TYPE EL3002_DEV_STATUS :
    STRUCT
      
		Underrange : BOOL;
		Overrange : BOOL;
		Limit1 : BOOL;
		Limit2 : BOOL;
		Error : BOOL;
		TxPDOState : BOOL;
		TxPDOToggle : BOOL;
	
    END_STRUCT
END_TYPE

(* stored: Version 1.1.0.1
   DUT EL3002_DEV_STATUS: Id {132520bd-724d-4855-8a18-6e5c4a322034} *)
